DATA_BLOCK "DB_HVAC_Live"
{ S7_Optimized_Access := 'FALSE' }
VERSION : 1.0
   STRUCT
      Data : "UDT_HVAC_Record";
   END_STRUCT;
BEGIN
END_DATA_BLOCK
